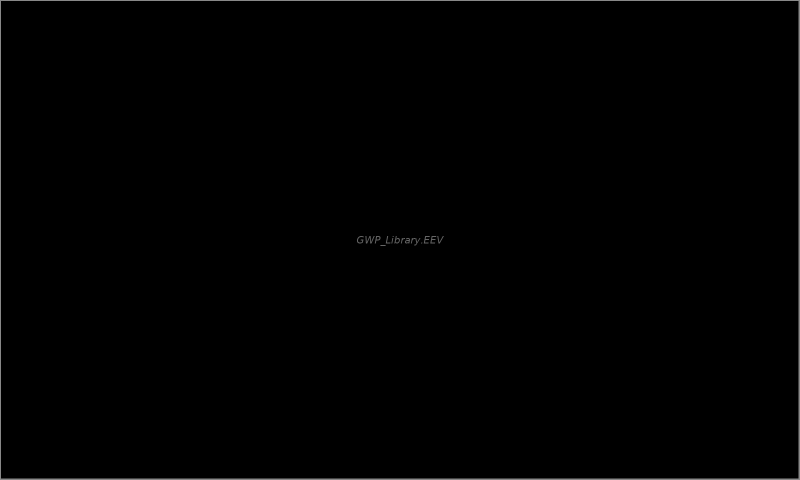
VISUALIZATION EEv  // 800x480
    Frame (0,0 800x480)
        shows GWP_Library.EEV(FB_EEV := Main.Kreis_3KO_0.EEV, FB_Init_1 := Main.Init_0)
END_VISUALIZATION

(* stored: Version 1.1.0.1, ProductVersion 3.1.4022.6
   Visu EEv: Id {e5bb20d3-55c9-4066-82ee-535d17fcb2d0} *)
